# EPICS autosave request: dxp/tags/R1-3beta2/iocBoot/iocDxpLinux_RC/auto_settings.req
file "mca_settings.req",                P=dxpLinux:, M=mca1
file "dxp_settings.req",                P=dxpLinux:, R=dxp1
